FUNCTION_BLOCK PUBLIC FB_ItalianPizzaPiccante EXTENDS FB_ItalianPizzaSalami
VAR_INPUT
END_VAR
VAR_OUTPUT
END_VAR
VAR
	bChilli		: BOOL := TRUE;
END_VAR

PROPERTY PUBLIC bHasChilli : BOOL
GET
bHasChilli := this^.bChilli;
END_GET
SET
this^.bChilli := bHasChilli;
END_SET
END_PROPERTY

METHOD PUBLIC GetPrice : LREAL
GetPrice := SUPER^.GetPrice();
IF (THIS^.bHasChilli) THEN
	GetPrice := GetPrice + 0.5;
END_IF
END_METHOD

END_FUNCTION_BLOCK

(* stored: Version 1.1.0.1, ProductVersion 3.1.4022.12
   POU FB_ItalianPizzaPiccante: Id {64337c8b-c5a9-4880-be10-7ff1e985eb1f}, SpecialFunc None
   Property bHasChilli: Id {df6ee347-b4bf-4978-9742-5976bc874d27}
   Get Get: Id {3bea9967-416f-4dd0-858d-153a0421a3b9}
   Set Set: Id {987be671-afd6-4bd4-a39f-8f21e145d49f}
   Method GetPrice: Id {6be45b42-fc6d-4f79-8b84-5c11df8741a7} *)
